Staubli VAL3: RecordExtAxis.pgx

public program RecordExtAxis(trsf& x_trTrsf, trsf& x_trPos, tool x_tTool)
  local jointRx l_jJ
  local pointRx l_pP
begin
  //  $recClean("c")
  //  $recAdd("c","CanIO\Axis8\posCmd_1")
  //  $recAdd("c","CanIO\Axis8\posFbk_1")
  //  $recStart("c",50,250)

  //  $recClean("c")
  //  $recAdd("c","extDrvCmdPos")
  //  $recAdd("c","extDrvCmdVel")
  //  $recAdd("c","extJntCmdPos")
  //  $recAdd("c","extJntCmdVel")
  //  $recAdd("c","extError")
  //  $recAdd("c","extDrvGrpError")
  //  $recStart("c",50,250)

 // x_pPos=$here
//    resize(nBuffSize,1,sel(x_b8Axis,2,1))
//  x_j=$XH(nBuffSize)
//  x_trTrsf.x=nBuffSize[0]
//  if x_b8Axis
//    x_trTrsf.y=nBuffSize[1]
//  endIf


if bMoveType
  $XframeLink(fFrame)
 l_pP=here(x_tTool,fFrame)
  x_trPos=l_pP.trsf

endIf




//记录七轴，八轴位置
call RecordJoint(l_jJ,x_trTrsf)




end
